// TwinCAT 3 PLC project Untitled1
// ProgramVersion: 3.1.4023.0
// libraries:
//   Tc2_Standard, * (Beckhoff Automation GmbH)
//   Tc2_System, * (Beckhoff Automation GmbH)
//   Tc3_Module, * (Beckhoff Automation GmbH)
// project tree:
//   / PlcTask.TcTTO
//   POUs/ MAIN.TcPOU
// real-time tasks:
//   TASK PlcTask: cycle T#10ms, priority 20, ADS port 350

CONFIGURATION Untitled1
    RESOURCE PLC ON TwinCAT3
        TASK PlcTask(INTERVAL := T#10ms, PRIORITY := 20);
        PROGRAM MAIN WITH PlcTask : MAIN;
    END_RESOURCE
END_CONFIGURATION

// ---- POUs/MAIN.TcPOU
PROGRAM MAIN
VAR
	FCS  : BOOL := FALSE;
	FCC : BOOL := FALSE;
	FCA  : BOOL := FALSE;
	FCB  : BOOL := FALSE;
	FC1 : BOOL := FALSE;
	FC2 : BOOL := FALSE;
	START  : BOOL := FALSE;
	RESET  : BOOL := FALSE;
	BRACCIOSUP  : BOOL := FALSE;
	BRACCIOINF : BOOL := FALSE;
	DX : BOOL := FALSE;
	SX : BOOL := FALSE;
	SU : BOOL := FALSE;
	GIU : BOOL := FALSE;
	CARICATO1 : BOOL := FALSE;
	CARICATO2 : BOOL := FALSE;
	M1 : BOOL := FALSE;
	M2 : BOOL := FALSE;
	P1 : BOOL := FALSE;
	P2 : BOOL := FALSE;
	G1 : BOOL := FALSE; //GIACCA
	G2 : BOOL := FALSE; //FELPA
	S1 : BOOL := FALSE;
	S2 : BOOL := FALSE;
	ALLARME : BOOL := FALSE;
	T_ALLARME : TIME := T#30S;
END_VAR

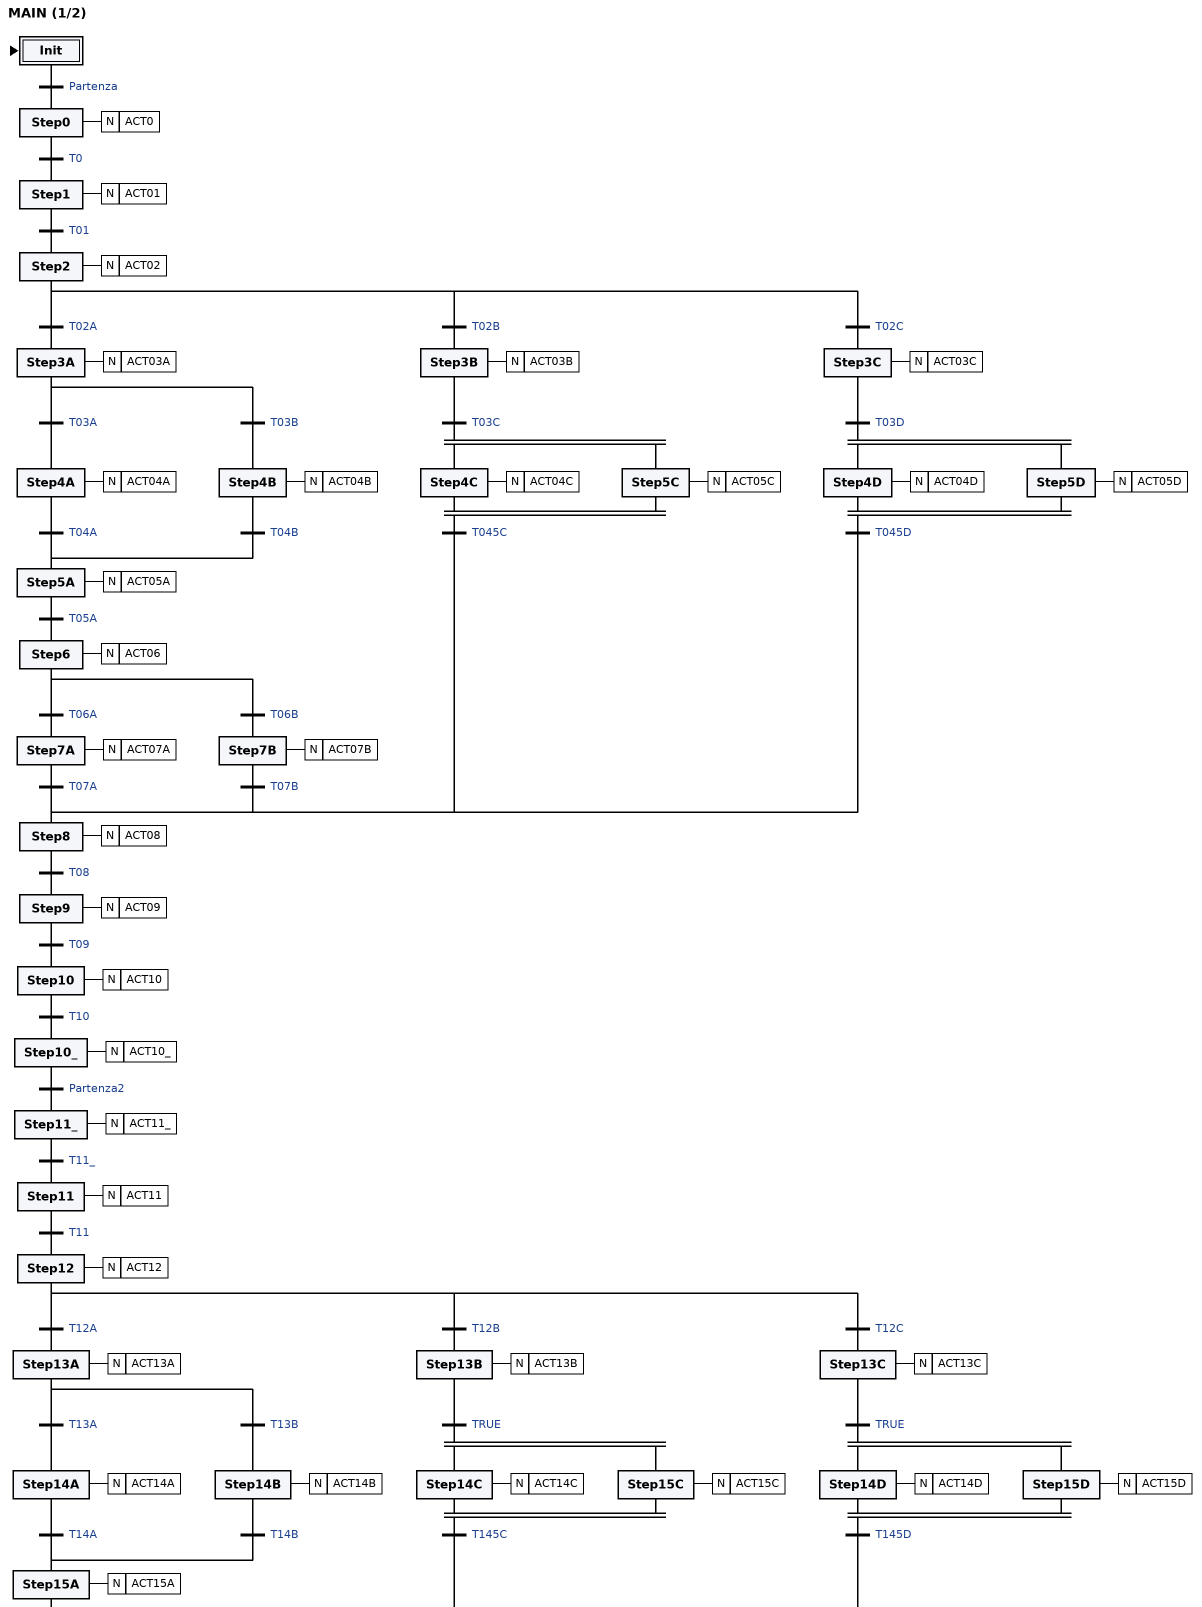
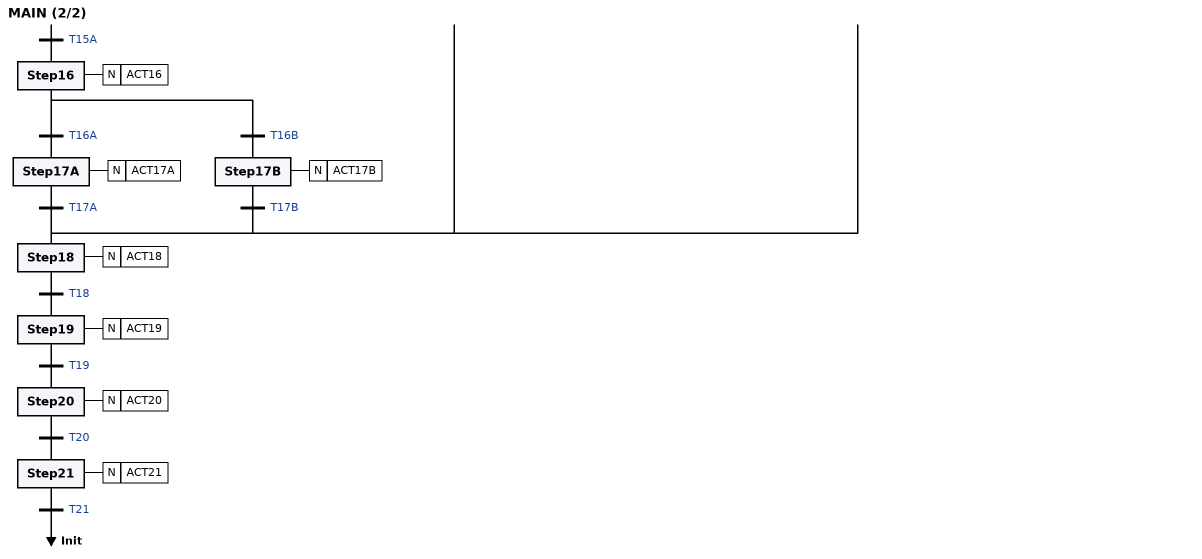
INITIAL_STEP Init:
END_STEP
TRANSITION FROM Init TO Step0
    := Partenza;
END_TRANSITION
STEP Step0:
    ACT0(N);
END_STEP
TRANSITION FROM Step0 TO Step1
    := T0;
END_TRANSITION
STEP Step1:
    ACT01(N);
END_STEP
TRANSITION FROM Step1 TO Step2
    := T01;
END_TRANSITION
STEP Step2:
    ACT02(N);
END_STEP
TRANSITION FROM Step2 TO Step3A
    := T02A;
END_TRANSITION
STEP Step3A:
    ACT03A(N);
END_STEP
TRANSITION FROM Step3A TO Step4A
    := T03A;
END_TRANSITION
STEP Step4A:
    ACT04A(N);
END_STEP
TRANSITION FROM Step4A TO Step5A
    := T04A;
END_TRANSITION
TRANSITION FROM Step3A TO Step4B
    := T03B;
END_TRANSITION
STEP Step4B:
    ACT04B(N);
END_STEP
TRANSITION FROM Step4B TO Step5A
    := T04B;
END_TRANSITION
STEP Step5A:
    ACT05A(N);
END_STEP
TRANSITION FROM Step5A TO Step6
    := T05A;
END_TRANSITION
STEP Step6:
    ACT06(N);
END_STEP
TRANSITION FROM Step6 TO Step7A
    := T06A;
END_TRANSITION
STEP Step7A:
    ACT07A(N);
END_STEP
TRANSITION FROM Step7A TO Step8
    := T07A;
END_TRANSITION
TRANSITION FROM Step6 TO Step7B
    := T06B;
END_TRANSITION
STEP Step7B:
    ACT07B(N);
END_STEP
TRANSITION FROM Step7B TO Step8
    := T07B;
END_TRANSITION
TRANSITION FROM Step2 TO Step3B
    := T02B;
END_TRANSITION
STEP Step3B:
    ACT03B(N);
END_STEP
TRANSITION FROM Step3B TO (Step4C, Step5C)
    := T03C;
END_TRANSITION
STEP Step4C:
    ACT04C(N);
END_STEP
STEP Step5C:
    ACT05C(N);
END_STEP
TRANSITION FROM (Step4C, Step5C) TO Step8
    := T045C;
END_TRANSITION
TRANSITION FROM Step2 TO Step3C
    := T02C;
END_TRANSITION
STEP Step3C:
    ACT03C(N);
END_STEP
TRANSITION FROM Step3C TO (Step4D, Step5D)
    := T03D;
END_TRANSITION
STEP Step4D:
    ACT04D(N);
END_STEP
STEP Step5D:
    ACT05D(N);
END_STEP
TRANSITION FROM (Step4D, Step5D) TO Step8
    := T045D;
END_TRANSITION
STEP Step8:
    ACT08(N);
END_STEP
TRANSITION FROM Step8 TO Step9
    := T08;
END_TRANSITION
STEP Step9:
    ACT09(N);
END_STEP
TRANSITION FROM Step9 TO Step10
    := T09;
END_TRANSITION
STEP Step10:
    ACT10(N);
END_STEP
TRANSITION FROM Step10 TO Step10_
    := T10;
END_TRANSITION
STEP Step10_:
    ACT10_(N);
END_STEP
TRANSITION FROM Step10_ TO Step11_
    := Partenza2;
END_TRANSITION
STEP Step11_:
    ACT11_(N);
END_STEP
TRANSITION FROM Step11_ TO Step11
    := T11_;
END_TRANSITION
STEP Step11:
    ACT11(N);
END_STEP
TRANSITION FROM Step11 TO Step12
    := T11;
END_TRANSITION
STEP Step12:
    ACT12(N);
END_STEP
TRANSITION FROM Step12 TO Step13A
    := T12A;
END_TRANSITION
STEP Step13A:
    ACT13A(N);
END_STEP
TRANSITION FROM Step13A TO Step14A
    := T13A;
END_TRANSITION
STEP Step14A:
    ACT14A(N);
END_STEP
TRANSITION FROM Step14A TO Step15A
    := T14A;
END_TRANSITION
TRANSITION FROM Step13A TO Step14B
    := T13B;
END_TRANSITION
STEP Step14B:
    ACT14B(N);
END_STEP
TRANSITION FROM Step14B TO Step15A
    := T14B;
END_TRANSITION
STEP Step15A:
    ACT15A(N);
END_STEP
TRANSITION FROM Step15A TO Step16
    := T15A;
END_TRANSITION
STEP Step16:
    ACT16(N);
END_STEP
TRANSITION FROM Step16 TO Step17A
    := T16A;
END_TRANSITION
STEP Step17A:
    ACT17A(N);
END_STEP
TRANSITION FROM Step17A TO Step18
    := T17A;
END_TRANSITION
TRANSITION FROM Step16 TO Step17B
    := T16B;
END_TRANSITION
STEP Step17B:
    ACT17B(N);
END_STEP
TRANSITION FROM Step17B TO Step18
    := T17B;
END_TRANSITION
TRANSITION FROM Step12 TO Step13B
    := T12B;
END_TRANSITION
STEP Step13B:
    ACT13B(N);
END_STEP
TRANSITION FROM Step13B TO (Step14C, Step15C)
    := TRUE;
END_TRANSITION
STEP Step14C:
    ACT14C(N);
END_STEP
STEP Step15C:
    ACT15C(N);
END_STEP
TRANSITION FROM (Step14C, Step15C) TO Step18
    := T145C;
END_TRANSITION
TRANSITION FROM Step12 TO Step13C
    := T12C;
END_TRANSITION
STEP Step13C:
    ACT13C(N);
END_STEP
TRANSITION FROM Step13C TO (Step14D, Step15D)
    := TRUE;
END_TRANSITION
STEP Step14D:
    ACT14D(N);
END_STEP
STEP Step15D:
    ACT15D(N);
END_STEP
TRANSITION FROM (Step14D, Step15D) TO Step18
    := T145D;
END_TRANSITION
STEP Step18:
    ACT18(N);
END_STEP
TRANSITION FROM Step18 TO Step19
    := T18;
END_TRANSITION
STEP Step19:
    ACT19(N);
END_STEP
TRANSITION FROM Step19 TO Step20
    := T19;
END_TRANSITION
STEP Step20:
    ACT20(N);
END_STEP
TRANSITION FROM Step20 TO Step21
    := T20;
END_TRANSITION
STEP Step21:
    ACT21(N);
END_STEP
TRANSITION FROM Step21 TO Init
    := T21;
END_TRANSITION
// branch label B01
// branch label B02
// branch label B03
// branch label B04

ACTION ACT0:
DX := TRUE;
END_ACTION

ACTION ACT01:
DX := FALSE;
SU := TRUE;
END_ACTION

ACTION ACT02:
SU := FALSE;
DX := TRUE;
END_ACTION

ACTION ACT03A:
DX := FALSE;
END_ACTION

ACTION ACT03B:
DX := FALSE;
END_ACTION

ACTION ACT03C:
DX := FALSE;
END_ACTION

ACTION ACT04A:
BRACCIOSUP := TRUE;
END_ACTION

ACTION ACT04B:
BRACCIOINF := TRUE;
END_ACTION

ACTION ACT04C:
BRACCIOSUP := TRUE;
END_ACTION

ACTION ACT04D:
BRACCIOSUP := TRUE;
END_ACTION

ACTION ACT05A:
DX := TRUE;
BRACCIOSUP := FALSE;
BRACCIOINF := FALSE;
END_ACTION

ACTION ACT05C:
BRACCIOINF := TRUE;
END_ACTION

ACTION ACT05D:
BRACCIOINF := TRUE;
END_ACTION

ACTION ACT06:
DX := FALSE;
END_ACTION

ACTION ACT07A:
BRACCIOSUP := TRUE;
END_ACTION

ACTION ACT07B:
BRACCIOINF := TRUE;
END_ACTION

ACTION ACT08:
SX := TRUE;
BRACCIOSUP := FALSE;
BRACCIOINF := FALSE;
END_ACTION

ACTION ACT09:
SX := FALSE;
GIU := TRUE;
END_ACTION

ACTION ACT10:
GIU := FALSE;
SX := TRUE;
END_ACTION

ACTION ACT10_:
SX := FALSE;
END_ACTION

ACTION ACT11:
GIU := TRUE;
DX := FALSE;
END_ACTION

ACTION ACT11_:
DX := TRUE;
END_ACTION

ACTION ACT12:
GIU := FALSE;
DX := TRUE;
END_ACTION

ACTION ACT13A:
DX := FALSE;
END_ACTION

ACTION ACT13B:
DX := FALSE;
END_ACTION

ACTION ACT13C:
DX := FALSE;
END_ACTION

ACTION ACT14A:
BRACCIOSUP := TRUE;
END_ACTION

ACTION ACT14B:
BRACCIOINF := TRUE;
END_ACTION

ACTION ACT14C:
BRACCIOSUP := TRUE;
END_ACTION

ACTION ACT14D:
BRACCIOSUP := TRUE;
END_ACTION

ACTION ACT15A:
DX := TRUE;
BRACCIOSUP := FALSE;
BRACCIOINF := FALSE;
END_ACTION

ACTION ACT15C:
BRACCIOINF := TRUE;
END_ACTION

ACTION ACT15D:
BRACCIOINF := TRUE;
END_ACTION

ACTION ACT16:
DX := FALSE;
END_ACTION

ACTION ACT17A:
BRACCIOSUP := TRUE;
END_ACTION

ACTION ACT17B:
BRACCIOINF := TRUE;
END_ACTION

ACTION ACT18:
SX := TRUE;
BRACCIOSUP := FALSE;
BRACCIOINF := FALSE;
END_ACTION

ACTION ACT19:
SX := FALSE;
SU := TRUE;
END_ACTION

ACTION ACT20:
SX := TRUE;
SU := FALSE;
END_ACTION

ACTION ACT21:
SX := FALSE;
END_ACTION

TRANSITION Partenza:
START AND ((M1 XOR M2) AND (P1 XOR P2)) ;
END_TRANSITION

TRANSITION Partenza2:
(NOT CARICATO1) AND (NOT CARICATO2) AND ((G1 XOR G2) AND (S1 XOR S2));
END_TRANSITION

TRANSITION T0:
FCC;
END_TRANSITION

TRANSITION T01:
FCA;
END_TRANSITION

TRANSITION T02A:
(FC1 AND (M1 XOR P1));
END_TRANSITION

TRANSITION T02B:
FC1 AND (M1 AND P1);
END_TRANSITION

TRANSITION T02C:
FC2 AND M2 AND P2;
END_TRANSITION

TRANSITION T03A:
M1;
END_TRANSITION

TRANSITION T03B:
P1;
END_TRANSITION

TRANSITION T03C:
TRUE;
END_TRANSITION

TRANSITION T03D:
TRUE;
END_TRANSITION

TRANSITION T045C:
CARICATO1 AND CARICATO2;
END_TRANSITION

TRANSITION T045D:
CARICATO1 AND CARICATO2;
END_TRANSITION

TRANSITION T04A:
CARICATO1;
END_TRANSITION

TRANSITION T04B:
CARICATO2;
END_TRANSITION

TRANSITION T05A:
FC2 AND (M2 OR P2);
END_TRANSITION

TRANSITION T06A:
M2;
END_TRANSITION

TRANSITION T06B:
P2;
END_TRANSITION

TRANSITION T07A:
CARICATO1;
END_TRANSITION

TRANSITION T07B:
CARICATO2;
END_TRANSITION

TRANSITION T08:
FCA;
END_TRANSITION

TRANSITION T09:
FCC;
END_TRANSITION

TRANSITION T10:
FCS;
END_TRANSITION

TRANSITION T11:
FCB;
END_TRANSITION

TRANSITION T11_:
FCC;
END_TRANSITION

TRANSITION T12A:
FC1 AND (G1 XOR S1)
END_TRANSITION

TRANSITION T12B:
FC1 AND (G1 AND S1);
END_TRANSITION

TRANSITION T12C:
FC2 AND (G2 AND S2);
END_TRANSITION

TRANSITION T13A:
G1;
END_TRANSITION

TRANSITION T13B:
S1;
END_TRANSITION

TRANSITION T145C:
CARICATO1 AND CARICATO2;
END_TRANSITION

TRANSITION T145D:
CARICATO1 AND CARICATO2;
END_TRANSITION

TRANSITION T14A:
CARICATO1;
END_TRANSITION

TRANSITION T14B:
CARICATO2;
END_TRANSITION

TRANSITION T15A:
FC2 AND (G2 XOR S2);
END_TRANSITION

TRANSITION T16A:
G2;
END_TRANSITION

TRANSITION T16B:
S2;
END_TRANSITION

TRANSITION T17A:
CARICATO1;
END_TRANSITION

TRANSITION T17B:
CARICATO2;
END_TRANSITION

TRANSITION T18:
FCB;
END_TRANSITION

TRANSITION T19:
FCC;
END_TRANSITION

TRANSITION T20:
FCS;
END_TRANSITION

TRANSITION T21:
(NOT CARICATO1) AND (NOT CARICATO2);
END_TRANSITION

END_PROGRAM
